FUNCTION_BLOCK fbSignalSimSliderWithGripper
VAR_IN_OUT
	em : ST_EM; 
END_VAR
VAR_INPUT
	EnableSim : BOOL;
	CmdSim : BOOL := true;
END_VAR
VAR
	 
	i : int; 
	delay: ARRAY [1..10] OF TON;
END_VAR

delay[1](PT:=T#2S); delay[1].ET;//Open GRIPPER Movement Sim
delay[2](PT:=T#2S); delay[2].ET;//Close GRIPPER Movement SIm
delay[3](PT:=T#5S); delay[3].ET;// Moving  PICK_POS //DROP_POS
delay[4](PT:=T#4S); delay[4].ET;//CMD.Clear simulation
delay[5](PT:=T#4S); delay[5].ET;
delay[6](PT:=T#4S); delay[6].ET;
delay[7](PT:=T#4S); delay[7].ET;//OpenGRipp State 0
delay[9](PT:=T#2S); delay[9].ET;//CMD.clear
delay[10](PT:=T#2S);delay[10].ET;//CMD.reset

IF EnableSim THEN
		
	IF em.Cmd = E_CMD.abort THEN
		delay[9](IN:=TRUE);
	END_IF
	
	IF em.Cmd = E_CMD.stop THEN
		delay[10](IN:=TRUE);
	END_IF
	
	
	
	CASE em.SequenceStep OF
		
		0:		//Undefined state
				
			
				//Simulate CMD.clear button
				
			IF delay[4].Q THEN
				delay[4](IN:=FALSE);
				em.Cmd:=E_CMD.reset;
			END_IF
			delay[4](IN:=TRUE);
				//Simulate movement to PICK_POS 
			IF em.Config.Data.Q[3]=TRUE THEN
				delay[3](IN:=TRUE);
			END_IF
			
			IF delay[3].Q THEN
					delay[3](IN:=FALSE);
					
					em.Config.Data.act_pos:=em.Config.Data.give_pos;	// Gripper position clear
					
			END_IF
	
			
			
			
		
		
		30:		//IDLE
				
				//WAIT FOR CMD					
			IF delay[6].Q THEN
				delay[6](IN:=FALSE);
				em.Cmd:=E_Cmd.start;
			END_IF
			delay[6](IN:=TRUE);
			
			
		40:		//EXECUTE.1
				
				//Simulate closing gripper
			IF em.Config.Data.Q[1]= TRUE THEN
				delay[2](IN:=TRUE);
			END_IF
			
			
			
			IF delay[2].Q THEN
				em.Config.Data.I[1]:= TRUE;
				em.Config.Data.I[2]:=FALSE;
				delay[2](IN:=FALSE);
			END_IF
		
	
		41:		//EXECUTE.2
				
			IF em.Config.Data.Q[3]=TRUE AND em.Config.Data.act_pos =em.Config.Data.pick_pos THEN  //servoGO		
				delay[3](IN:=TRUE);	
				em.Config.Data.act_pos:=666; //LEAVING HOME
			END_IF
				
			IF delay[3].Q THEN
				delay[3].IN:=FALSE;
				em.Config.Data.act_pos:= em.Config.Data.give_pos;		
			END_IF
		
		
		42:		//EXECUTE.3 OPEN GRIPPER
		
				//Simulate opening gripper
			IF em.Config.Data.Q[1]= FALSE  THEN
			delay[1](IN:=TRUE);
			
			END_IF
	 
			IF delay[1].Q THEN
				em.Config.Data.I[1]:= FALSE;
				em.Config.Data.I[2]:=TRUE;
				delay[1](IN:=FALSE);
			END_IF
		43:		//EXECUTE.4 MOVING PICK_pOS 
		
			IF em.Config.Data.Q[3]=TRUE AND
			em.Config.Data.act_pos =em.Config.Data.drop_pos THEN
				delay[3](IN:=TRUE);	
				em.Config.Data.act_pos:=666;
			END_IF
				
			IF delay[3].Q THEN
			delay[3].IN:=FALSE;
			em.Config.Data.act_pos:=em.Config.Data.give_pos; // arrived at pick_pos
			END_IF;
				
		65:		//ABORTED
		
			IF delay[9].Q THEN
			delay[9].IN:=FALSE;
			em.Cmd:=E_Cmd.clear;
			delay[10].IN:=TRUE;
			END_IF
		
		
		70:		//STOPPED
			IF delay[10].Q THEN
			delay[10].IN:=FALSE;
			em.Cmd:=E_Cmd.reset;
			END_IF
	END_CASE
	
END_IF

END_FUNCTION_BLOCK

(* stored: Version 1.1.0.1, ProductVersion 3.1.4024.12
   POU fbSignalSimSliderWithGripper: Id {e37b1043-ba32-4968-85cd-3c6e65122a2b}, SpecialFunc None *)
